{attribute 'qualified_only'}
VAR_GLOBAL
END_VAR

(* stored: Version 1.1.0.1
   GVL GVL_HIKROBOT_COMMANDS: Id {ef3780e1-11eb-4099-badb-6bd7ab8e3a98} *)
